// TIA Portal V18 export
TYPE "UDT_HCsAO"
// stored: IsFailsafeCompliant false
   STRUCT
      rHC3vwCtrl : Array[1..2] of Real;
   END_STRUCT;
END_TYPE
